{attribute 'GeneratedUsingTerminal: EK1100-0000-0018'}
{attribute addProperty BoxType "EK1100-0000-0018"}
{attribute addProperty Id "Beckhoff_EJ4xxxEK1122Beckhoff_EJ4xxxEK1122_E11BF0B62A_0001_EJ4002_0000_0017EJ4002_EE36E02D7A_0002_EJ4002_0000_0018EJ4002_D295D1387A_0003_EJ4004_0000_0020EJ4004_4A1E805A11A_0004_EJ4008_0000_0020EJ4008_255938B619A_0005_EJ4018_0000_0016EJ4018_255938B619A_0006_EJ4024_0000_0020EJ4024_4A1E805A11A_0007_EJ4132_0000_0019EJ4132_EE36E02D7A_0008_EJ4134_0000_0019EJ4134_57A43C6411A_0009_EJ4134_0000_0020EJ4134_57A43C6411"}
{attribute addProperty CRC "436561731"}
{attribute addProperty Size "105"}
TYPE Beckhoff_EJ4xxx_1A056743 EXTENDS EK1100_1FC0878B :
STRUCT
	{attribute addProperty Name "Beckhoff_EJ4xxxEK1122"}
	{attribute addProperty PreviousPort "Beckhoff EJ4xxx : B"}
	Beckhoff_EJ4xxxEK1122 : Beckhoff_EJ4xxxEK1122_E11BF0B6;
	{attribute addProperty Name "A_0001_EJ4002_0000_0017"}
	{attribute addProperty PreviousPort "Beckhoff EJ4xxxEK1122 : C"}
	A_0001_EJ4002_0000_0017 : EJ4002_EE36E02D;
	{attribute addProperty Name "A_0002_EJ4002_0000_0018"}
	{attribute addProperty PreviousPort "A_0001(EJ4002-0000-0017) : B"}
	A_0002_EJ4002_0000_0018 : EJ4002_D295D138;
	{attribute addProperty Name "A_0003_EJ4004_0000_0020"}
	{attribute addProperty PreviousPort "A_0002(EJ4002-0000-0018) : B"}
	A_0003_EJ4004_0000_0020 : EJ4004_4A1E805A;
	{attribute addProperty Name "A_0004_EJ4008_0000_0020"}
	{attribute addProperty PreviousPort "A_0003(EJ4004-0000-0020) : B"}
	A_0004_EJ4008_0000_0020 : EJ4008_255938B6;
	{attribute addProperty Name "A_0005_EJ4018_0000_0016"}
	{attribute addProperty PreviousPort "A_0004(EJ4008-0000-0020) : B"}
	A_0005_EJ4018_0000_0016 : EJ4018_255938B6;
	{attribute addProperty Name "A_0006_EJ4024_0000_0020"}
	{attribute addProperty PreviousPort "A_0005(EJ4018-0000-0016) : B"}
	A_0006_EJ4024_0000_0020 : EJ4024_4A1E805A;
	{attribute addProperty Name "A_0007_EJ4132_0000_0019"}
	{attribute addProperty PreviousPort "A_0006(EJ4024-0000-0020) : B"}
	A_0007_EJ4132_0000_0019 : EJ4132_EE36E02D;
	{attribute addProperty Name "A_0008_EJ4134_0000_0019"}
	{attribute addProperty PreviousPort "A_0007(EJ4132-0000-0019) : B"}
	A_0008_EJ4134_0000_0019 : EJ4134_57A43C64;
	{attribute addProperty Name "A_0009_EJ4134_0000_0020"}
	{attribute addProperty PreviousPort "A_0008(EJ4134-0000-0019) : B"}
	A_0009_EJ4134_0000_0020 : EJ4134_57A43C64;
END_STRUCT
END_TYPE

(* stored: Version 1.2.0.0, ProductVersion 3.1.4024.9
   DUT Beckhoff_EJ4xxx_1A056743: Id {7ce48b3b-a03b-4607-bf15-ce47869adc41} *)
